(* CoDeSys 2.3.9.50 project: CX8051 HJCS 20.8.22.pro *)
(* Libraries: STANDARD.LIB 5.6.98 12:03:02 *)

(* Task configuration *)
TASK Standard (PRIORITY := 0, INTERVAL := T#10ms);
	MAIN
END_TASK

(* Global variable list: TwinCAT_Configuration *)
(* Generated automatically by TwinCAT - (read only) *)
VAR_CONFIG
	MAIN.CAN_OUT AT %QB0 : ARRAY [1..16] OF BYTE;
	MAIN.CAN_IN AT %IB0 : ARRAY [1..16] OF BYTE;
	MAIN.EtherCAT_OUT AT %QB16 : ARRAY [1..16] OF BYTE;
	MAIN.EtherCAT_IN AT %IB16 : ARRAY [1..16] OF BYTE;
END_VAR

(* POU MAIN, ST *)
PROGRAM MAIN
VAR

	CAN_OUT AT %Q*: ARRAY [1..16]  OF BYTE;

	CAN_IN  AT %I*:ARRAY [1..16]  OF BYTE ;

	EtherCAT_OUT AT %Q*: ARRAY [1..16]  OF BYTE;

	EtherCAT_IN  AT %I*:ARRAY [1..16]  OF BYTE ;

        x1:BOOL;
END_VAR
EtherCAT_OUT[1].1:=1;

EtherCAT_OUT[2].0:=CAN_IN [2].1;

EtherCAT_OUT[2].1:=CAN_IN [2].2;

EtherCAT_OUT[2].2:=CAN_IN [2].3

;
END_PROGRAM
